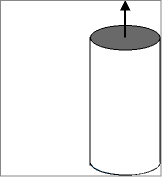
VISUALIZATION VISU_Tube_Top_11  // 162x177
VAR_IN_OUT
	azi : LREAL;
END_VAR
    Ellipse (90,150 70x25)
        p2858320360: azi
    Polygon (90,35) (160,35) (160,162) (157,167) (155,168) (149,171) (142,173) (135,174) (127,174) (119,174) (111,173) (102,171) (94,167) (90,162)
        p2858320360: azi
    Ellipse (90,25 70x25)
        p2858320360: azi
    Polygon (120,10) (125,0) (130,10)
        p2858320360: azi
    Polyline (125,37) (125,10)
        p2858320360: azi
    Polyline (90,165) (90,37)
        p2858320360: azi
    Polyline (160,162) (160,37)
        p2858320360: azi
END_VISUALIZATION

(* stored: Version 1.1.0.1, ProductVersion 3.1.4018.5
   Visu VISU_Tube_Top_11: Id {1b7305ac-3338-4cf7-82bb-75be8f0fdabd} *)
